(*
Used to request a beam parameter set from EPICS.

Technically just one of these is needed in the entire
PMPS for a line.

*)
FUNCTION_BLOCK FB_BPControlDevice
VAR_INPUT
END_VAR
VAR_OUTPUT
END_VAR
VAR_IN_OUT
	Arbiter : FB_Arbiter;
END_VAR
VAR
	{attribute 'pytmc' := '
    	pv: ReqBP
		io: o
    '}
	EpicsReqBP : ST_BeamParams;
	{attribute 'pytmc' := '
    	pv: Apply
		io: o
    '}
	bApply : BOOL;
	
	nControlDeviceID : DWORD;
	
	rtApply : R_TRIG;
	
END_VAR


rtApply(CLK:=bApply);
IF rtApply.Q THEN
	Arbiter.RemoveRequest(nControlDeviceID);
	Arbiter.AddRequest(nControlDeviceID, EpicsReqBP);
	bApply := FALSE;
END_IF

METHOD FB_init : BOOL
VAR_INPUT
	bInitRetains : BOOL; // if TRUE, the retain variables are initialized (warm start / cold start)
	bInCopyCode : BOOL;  // if TRUE, the instance afterwards gets moved into the copy code (online change)
	nID : DWORD := PMPS_GVL.EXCLUDED_ASSERTION_ID;
END_VAR
nControlDeviceID:= nID;
END_METHOD

END_FUNCTION_BLOCK

(* stored: Version 1.1.0.1, ProductVersion 3.1.4022.18
   POU FB_BPControlDevice: Id {c3303296-37d2-4688-9929-f388bfe14617}, SpecialFunc None
   Method FB_init: Id {d7dd8caa-2a9b-478e-8c53-254b06d26293} *)
